Universal Robots PolyScope program: Group21Lab1Task1.urp

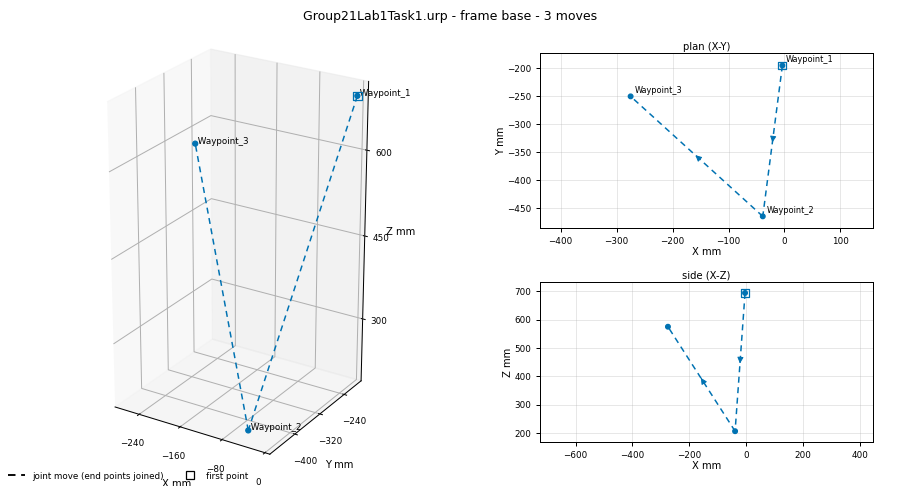
[picture p0: tool path of Group21Lab1Task1.urp in frame base, 3 of 3 moves have a stored position in this frame; points joined in program order, loops and branches not executed]
Program grou21 (createdIn=3.5.0.10584 lastSavedIn=3.5.0.10584 directory=/programs/usbdisk installation=default robotSerialNumber=2017332505)
Calibrated DH parameters: a=[0, -0.24355, -0.210285, 0.000007, -0.000026, 0]; d=[0.151972, 1.341373, 3.010199, -4.239311, 0.085317, 0.082321]; alpha=[1.570715, -0.004846, 0.008121, 1.57079, -1.571065, 0]; deltaTheta=[0.000017, -0.02667, 0.193133, -0.166555, -0.000046, 0.000042]
Robot Program (runOnlyOnce=false motionType=MoveJ speed=1.047198 acceleration=1.396263 useActiveTCP=false)
  MoveJ speed 60 deg/s, acceleration 80 deg/s^2 (useActiveTCP=false)
    Waypoint Waypoint_1: TCP in base x=-3.769 y=-194.843 z=693.855 mm, rx=0 ry=-0.0063 rz=-0.001 rad; joints [-0.018, -89.667, -0.136, -89.511, 0.051, -0.417] deg
    Waypoint Waypoint_2: TCP in base x=-38.818 y=-464.442 z=207.454 mm, rx=1.4939 ry=0.0767 rz=0.065 rad; joints [70.863, -50.349, 65.498, -109.303, -88.695, -23.986] deg
    Waypoint Waypoint_3: TCP in base x=-275.044 y=-249.982 z=574.983 mm, rx=1.2001 ry=1.2 rz=-1.2 rad; joints [31.247, -59.656, 22.56, -142.246, -120.837, -88.995] deg; flange x=-275 y=-250 z=575 mm, rx=-0.0001 ry=-1.5784 rz=0.0119 rad
